(* CODESYS project 3 Automatic Grinding Process.project

Project tree, tasks and I/O mapping:
  Device : CODESYS Control Win V3, 3S - Smart Software Solutions GmbH, order no. 305021, version 3.5.7.0
    application Application
      libraries: Standard, * (System)
      task MainTask (cyclic, interval t#20ms, priority 1) calls PLC_PRG
      task VISU_TASK (cyclic, interval 100 ms, priority 31) calls VisuElems.Visu_Prg
      program PLC_PRG [LD]
      visualisation Visualization
  text list GlobalTextList
*)

// Device/Application/PLC_PRG
PROGRAM PLC_PRG
VAR
	TON_01: TON;
	start: BOOL;
	stop: BOOL;
	start_latch: BOOL;
	job_in_sensor: BOOL;
	job_out_sensor: BOOL;
	job_sensor_latch: BOOL;
	fine_sensor_memory: BOOL;
	rough_sensor_memory: BOOL;
	conveyor_motor: BOOL;
	TON_02: TON;
	rough_sensor: BOOL;
	fine_sensor: BOOL;
	rough_grinding_motor: BOOL;
	TTT: TIME;
	fine_grinding_motor: BOOL;
	packing_session: BOOL;
	TTTT: TIME;
END_VAR
VAR // added by the converter: edge detectors and wires of the graphical bodies
    _w1, _w2 : BOOL;
END_VAR

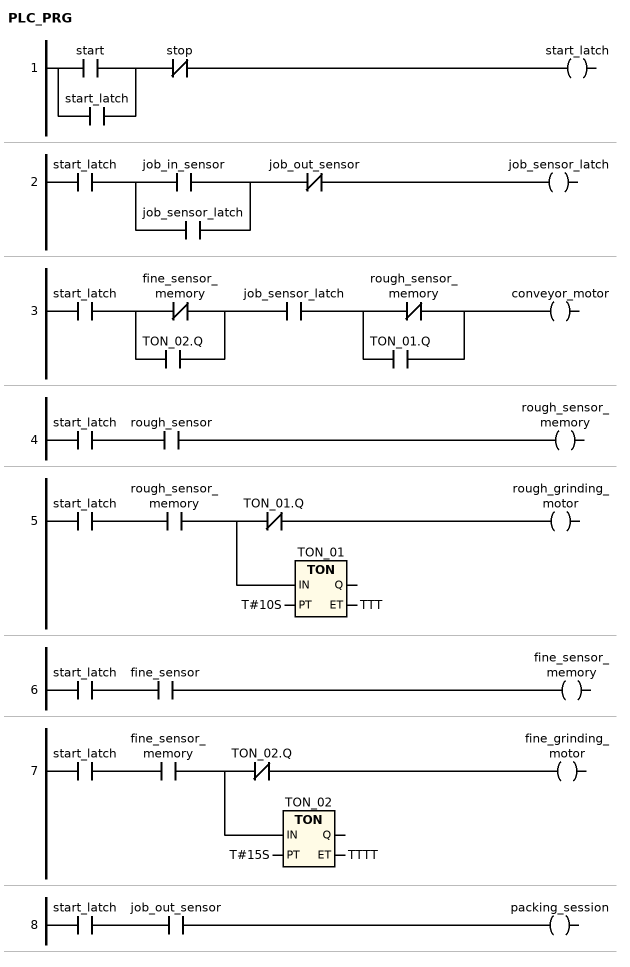
// NETWORK 1
start_latch := (start OR start_latch) AND NOT stop;

// NETWORK 2
job_sensor_latch := start_latch AND (job_in_sensor OR job_sensor_latch) AND NOT job_out_sensor;

// NETWORK 3
conveyor_motor := start_latch AND (NOT fine_sensor_memory OR TON_02.Q) AND job_sensor_latch AND (NOT rough_sensor_memory OR TON_01.Q);

// NETWORK 4
rough_sensor_memory := start_latch AND rough_sensor;

// NETWORK 5
_w1 := start_latch AND rough_sensor_memory;
rough_grinding_motor := _w1 AND NOT TON_01.Q;
TON_01(IN := _w1, PT := T#10S, ET => TTT); // TON

// NETWORK 6
fine_sensor_memory := start_latch AND fine_sensor;

// NETWORK 7
_w2 := start_latch AND fine_sensor_memory;
fine_grinding_motor := _w2 AND NOT TON_02.Q;
TON_02(IN := _w2, PT := T#15S, ET => TTTT); // TON

// NETWORK 8
packing_session := start_latch AND job_out_sensor;

END_PROGRAM

// Device/Application/Visualization
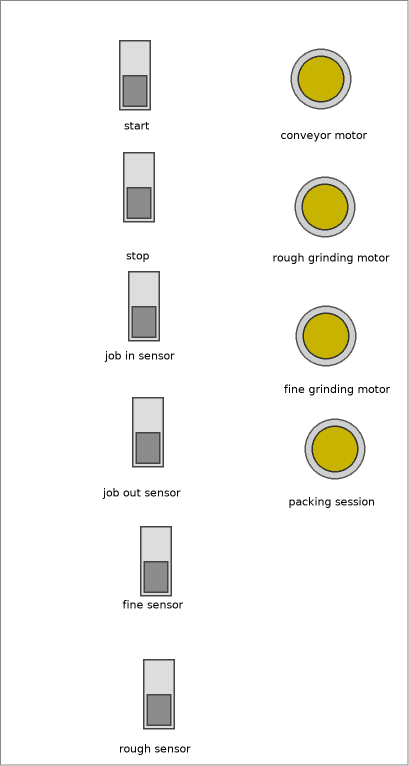
VISUALIZATION Visualization  // 409x766
    DipSwitch (100,40 70x70), variable: PLC_PRG.start, behaviour: TOGGLE, style: Switch-DipSwitch-Gray
    DipSwitch (104,152 70x70), variable: PLC_PRG.stop, behaviour: TOGGLE, style: Switch-DipSwitch-Gray
    DipSwitch (109,271 70x70), variable: PLC_PRG.job_in_sensor, behaviour: TOGGLE, style: Switch-DipSwitch-Gray
    DipSwitch (113,397 70x70), variable: PLC_PRG.job_out_sensor, behaviour: TOGGLE, style: Switch-DipSwitch-Gray
    DipSwitch (121,526 70x70), variable: PLC_PRG.fine_sensor, behaviour: TOGGLE, style: Switch-DipSwitch-Gray
    DipSwitch (124,659 70x70), variable: PLC_PRG.rough_sensor, behaviour: TOGGLE, style: Switch-DipSwitch-Gray
    Lamp1 (286,44 70x70), variable: PLC_PRG.conveyor_motor, style: Lamp-Lamp1-Yellow
    Lamp1 (290,172 70x70), variable: PLC_PRG.rough_grinding_motor, style: Lamp-Lamp1-Yellow
    Lamp1 (291,301 70x70), variable: PLC_PRG.fine_grinding_motor, style: Lamp-Lamp1-Yellow
    Lamp1 (300,414 70x70), variable: PLC_PRG.packing_session, style: Lamp-Lamp1-Yellow
    Label (62,111 150x30), "start"
    Label (260,111 128x49), "conveyor motor"
    Label (63,241 150x30), "stop"
    Label (256,243 150x30), "rough grinding motor"
    Label (269,373 136x33), "fine grinding motor"
    Label (65,341 150x30), "job in sensor"
    Label (67,478 150x30), "job out sensor"
    Label (257,487 150x30), "packing session"
    Label (78,590 150x30), "fine sensor"
    Label (80,734 150x30), "rough sensor"
END_VISUALIZATION
